(* for use with EtherCAT temperature sensor terminals *)
FUNCTION_BLOCK FB_EBUS_TempSensor
VAR_INPUT
	bEnable				: BOOL;		(* TRUE = enable sensor monitoring *)
	bReset				: BOOL;		(* TRUE = reset sensor error *)
	sEtherCATState		: ST_EBUS_EtherCATState;	(* EtherCAT operating state *)
	sDataIn				: ST_EBUS_AnalogueDataIn;	(* input data *)
END_VAR
VAR_OUTPUT
	bStatusOK			: BOOL;		(* comms and sensor status OK *)
	bError				: BOOL;		(* sensor error active *)
	fTemperature		: LREAL;		(* temperature in degC *)
END_VAR
VAR
	bCommsStatusOK		: BOOL;
	fbError				: SR;
END_VAR
(*
-------------------------------------------------------------------------------------------------
Date		Version	Author	Comments
-------------------------------------------------------------------------------------------------
30/01/2015	3.00.00	PB		Updated to use ST_EBUS_EtherCATState and ST_EBUS_AnalogueDataIn
							All floating point values now use LREAL

-------------------------------------------------------------------------------------------------
13/04/2010	1.02.01	PB		Bug fix - bCommsStatusOK now uses EtherCAT State = 8 instead of 0 
31/03/2010	1.02.00	PB		Initial release
-------------------------------------------------------------------------------------------------
*)

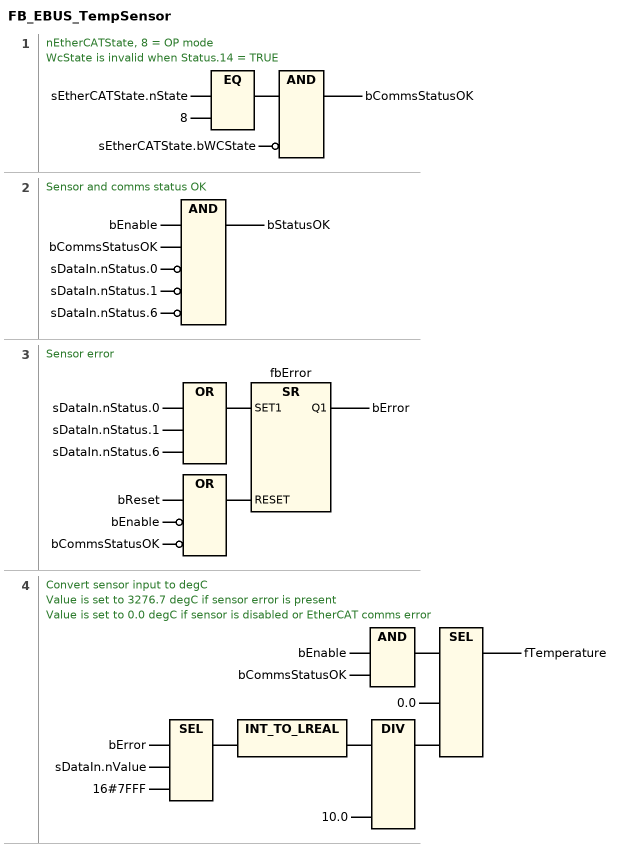
// NETWORK 1
// 					nEtherCATState, 8 = OP mode
// WcState is invalid when Status.14 = TRUE
//
bCommsStatusOK := sEtherCATState.nState = 8 AND NOT sEtherCATState.bWCState;

// NETWORK 2
// Sensor and comms status OK
bStatusOK := bEnable AND bCommsStatusOK AND NOT sDataIn.nStatus.0 AND NOT sDataIn.nStatus.1 AND NOT sDataIn.nStatus.6;

// NETWORK 3
// Sensor error
fbError(SET1 := sDataIn.nStatus.0 OR sDataIn.nStatus.1 OR sDataIn.nStatus.6, RESET := bReset OR NOT bEnable OR NOT bCommsStatusOK); // SR
bError := fbError.Q1;

// NETWORK 4
// 					Convert sensor input to degC
// Value is set to 3276.7 degC if sensor error is present
// Value is set to 0.0 degC if sensor is disabled or EtherCAT comms error
//
//
fTemperature := SEL(bEnable AND bCommsStatusOK, 0.0, INT_TO_LREAL(SEL(bError, sDataIn.nValue, 16#7FFF)) / 10.0);

END_FUNCTION_BLOCK

(* stored: Version 1.1.0.1, ProductVersion 3.1.4024.15
   POU FB_EBUS_TempSensor: Id {9abae6e3-df28-4d33-99c1-85b019596989}, SpecialFunc None *)
